PROGRAM Reset
VAR
END_VAR

END_PROGRAM

(* stored: Version 1.1.0.1, ProductVersion 3.1.4024.12
   POU Reset: Id {e7d61cc6-e7cc-498a-bbe3-a4a9af06d679}, SpecialFunc None *)
